SYSTEM LIFTER_VIEWL (* Lifter with Feed & Takeoff Conveyors *)
  (* Standard: 61499-1; Classification: Simulation; ApplicationDomain: Assembly; Type: Dual Stroke Cylinder *)
  (* Version 0.1, 2004-12-19, JHC, Rockwell Automation, Adjusted frame heights for WinXP. *)
  (* Version 0.0, 2004-06-10, JHC, Rockwell Automation, Adapted from DRILL_VIEWL *)
  DEVICE HMI : FRAME_DEVICE(BOUNDS := [100,100,350,205], GRID := [1,1])
    RESOURCE RES1 : PANEL_RESOURCE
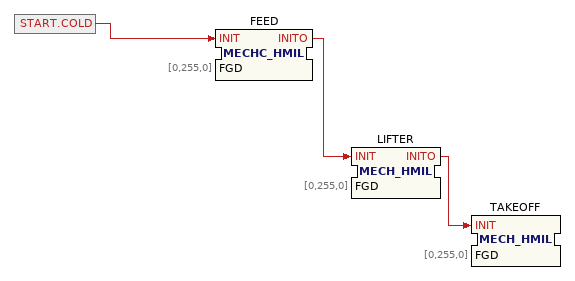
      FBS
        TAKEOFF : MECH_HMIL(FGD := [0,255,0]);
        FEED : MECHC_HMIL(FGD := [0,255,0]);
        LIFTER : MECH_HMIL(FGD := [0,255,0]);
      END_FBS
      EVENT_CONNECTIONS
        START.COLD TO FEED.INIT;
        LIFTER.INITO TO TAKEOFF.INIT;
        FEED.INITO TO LIFTER.INIT;
      END_CONNECTIONS
    END_RESOURCE
  END_DEVICE
  DEVICE VIEW : FRAME_DEVICE(BOUNDS := [450,100,160,205])
    RESOURCE LIFTER : VIEW_PANEL(DIA := 30, SIZE := [5,5], VERTICAL := 1)
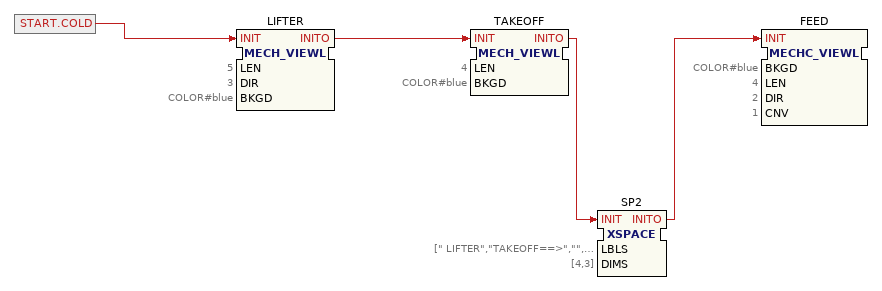
      FBS
        LIFTER : MECH_VIEWL(LEN := 5, DIR := 3, BKGD := COLOR#blue);
        FEED : MECHC_VIEWL(BKGD := COLOR#blue, LEN := 4, DIR := 2, CNV := 1); (* Feed Conveyor *)
        SP2 : XSPACE(LBLS := [" LIFTER","TAKEOFF==>","","<==FEED"], DIMS := [4,3]);
        TAKEOFF : MECH_VIEWL(LEN := 4, BKGD := COLOR#blue); (* Takeoff Conveyor *)
      END_FBS
      EVENT_CONNECTIONS
        TAKEOFF.INITO TO SP2.INIT;
        SP2.INITO TO FEED.INIT;
        START.COLD TO LIFTER.INIT;
        LIFTER.INITO TO TAKEOFF.INIT;
      END_CONNECTIONS
    END_RESOURCE
  END_DEVICE
END_SYSTEM
